(* IEC 61131-3 sources: Lasal/CPU_5344_V01/Class/Ifm2330Output, 1 file *)

(* ---- Ifm2330Output.st ---- *)
(*!
<Class
	Name               = "Ifm2330Output"
	Revision           = "0.0"
	RealtimeTask       = "false"
	CyclicTask         = "true"
	DefCyclictime      = "2 ms"
	BackgroundTask     = "false"
	Sigmatek           = "false"
	OSInterface        = "false"
	HighPriority       = "false"
	Automatic          = "false"
	UpdateMode         = "Prescan"
	SharedCommandTable = "true"
	Objectsize         = "(660,960)">
	<Channels>
		<Server Name="ActualMode" Visualized="true" Remotely="true" Initialize="false" WriteProtected="true" Retentive="false" Comment="Shows the currently active mode of the device (is only valid when the ClassState is _ClassOk and the FaultFlags are on _NoFault)"/>
		<Server Name="ClassState" Class="SDCIDevice" Visualized="true" Remotely="true" Initialize="false" WriteProtected="true" Retentive="false" Comment="Shows the current Status of the Hardware Class"/>
		<Server Name="ClassSvr" Visualized="false" Initialize="false" WriteProtected="true" Retentive="false"/>
		<Server Name="Output1" Visualized="false" Initialize="false" WriteProtected="false" Retentive="false"/>
		<Server Name="Output10" Visualized="false" Initialize="false" WriteProtected="false" Retentive="false"/>
		<Server Name="Output11" Visualized="false" Initialize="false" WriteProtected="false" Retentive="false"/>
		<Server Name="Output12" Visualized="false" Initialize="false" WriteProtected="false" Retentive="false"/>
		<Server Name="Output2" Visualized="false" Initialize="false" WriteProtected="false" Retentive="false"/>
		<Server Name="Output3" Visualized="false" Initialize="false" WriteProtected="false" Retentive="false"/>
		<Server Name="Output4" Visualized="false" Initialize="false" WriteProtected="false" Retentive="false"/>
		<Server Name="Output5" Visualized="false" Initialize="false" WriteProtected="false" Retentive="false"/>
		<Server Name="Output6" Visualized="false" Initialize="false" WriteProtected="false" Retentive="false"/>
		<Server Name="Output7" Visualized="false" Initialize="false" WriteProtected="false" Retentive="false"/>
		<Server Name="Output8" Visualized="false" Initialize="false" WriteProtected="false" Retentive="false"/>
		<Server Name="Output9" Visualized="false" Initialize="false" WriteProtected="false" Retentive="false"/>
		<Client Name="SDCIClass" Required="true" Internal="true"/>
		<Client Name="SdciIn" Required="false" Internal="false"/>
	</Channels>
	<Network Name="Ifm2330Output">
		<!-- List of Components in this network -->
		<Components>
			<Object
				Name       = "SDCIClass"
				Class      = "SDCIClassIFM2330"
				Position   = "(150,120)"
				Visualized = "true"
				Remotely   = "true">
				<Channels>
					<Server Name="ActualMode"/>
					<Server Name="ClassState"/>
					<Server Name="DeviceID"/>
					<Server Name="DirectInput"/>
					<Server Name="FaultFlags"/>
					<Server Name="Input"/>
					<Server Name="MinCycleTime"/>
					<Server Name="NbrOfEventsAvailable"/>
					<Server Name="Output"/>
					<Server Name="PortStateBits"/>
					<Server Name="VendorID"/>
					<Client Name="ReadPdoSize" Value="64"/>
					<Client Name="Required" Value="0"/>
					<Client Name="SdciIn"/>
					<Client Name="SkipEndianSwap" Value="0"/>
					<Client Name="StartUpMode" Value="_SDCI"/>
					<Client Name="WritePdoSize" Value="32"/>
				</Channels>
				<AdditionalData>
					<Entry Name="DeviceType" Value="SDCIClassIFM2330"/>
				</AdditionalData>
			</Object>
		</Components>
		<Comments>
		</Comments>
		<!-- List of Connections in this network -->
		<Connections>
			<Connection Source="SDCIClass.SdciIn" Destination="this.SdciIn" Vertices="(150,210),(38,210),"/>
			<Connection Source="this.ClassState" Destination="SDCIClass.ClassState" Vertices="(990,270),(818,210),"/>
			<Connection Source="this.SDCIClass" Destination="SDCIClass.ClassState"/>
			<Connection Source="this.ActualMode" Destination="SDCIClass.ActualMode" Vertices="(990,330),(818,450),"/>
		</Connections>
		<!-- Headerfiles -->
		<Options>
		</Options>
	</Network>
</Class>
*)
Ifm2330Output : CLASS
  //Servers:
	ClassSvr 	: SvrChCmd_DINT;
	ClassState 	: SvrChCmd_t_e_VaranErrors;
	ActualMode 	: SvrCh_t_SDCIPortMode_PTofCls_SdiasSDCIMaster;
	Output1 	: SvrCh_DINT;
	Output2 	: SvrCh_DINT;
	Output3 	: SvrCh_DINT;
	Output4 	: SvrCh_DINT;
	Output5 	: SvrCh_DINT;
	Output6 	: SvrCh_DINT;
	Output7 	: SvrCh_DINT;
	Output8 	: SvrCh_DINT;
	Output9 	: SvrCh_DINT;
	Output10 	: SvrCh_DINT;
	Output11 	: SvrCh_DINT;
	Output12 	: SvrCh_DINT;
  //Clients:
	SdciIn 	: CltChCmd_DINT;
	SDCIClass 	: CltChCmd_SDCIClassIFM2330;
  //Variables:
		bdOutputs : BDINT
		[
		];

  //Functions:

	FUNCTION VIRTUAL GLOBAL Init;

	FUNCTION VIRTUAL GLOBAL CyWork
		VAR_INPUT
			EAX 	: UDINT;
		END_VAR
		VAR_OUTPUT
			state (EAX) 	: UDINT;
		END_VAR;

	FUNCTION VIRTUAL GLOBAL ClassState::Read
		VAR_OUTPUT
			output (EAX) 	: t_e_VaranErrors;
		END_VAR;

	FUNCTION VIRTUAL GLOBAL ActualMode::Read
		VAR_OUTPUT
			output (EAX) 	: SdiasSDCIMaster::t_SDCIPortMode;
		END_VAR;
  //Tables:
	FUNCTION @STD
		VAR_OUTPUT
			ret_code	: CONFSTATES;
		END_VAR;
	FUNCTION GLOBAL TAB @CT_;
END_CLASS;

#pragma using SDCIClassIFM2330

//avdb 29092017 outputs io eiland IFM

FUNCTION VIRTUAL GLOBAL Ifm2330Output::CyWork
	VAR_INPUT
		EAX 	: UDINT;
	END_VAR
	VAR_OUTPUT
		state (EAX) 	: UDINT;
	END_VAR

  // get outputs from servers
  bdOutputs.25 := Output1=1;
  bdOutputs.9 := Output2=1;
  bdOutputs.17 := Output3=1;
  bdOutputs.1 := Output4=1;
  bdOutputs.26 := Output5=1;
  bdOutputs.10 := Output6=1;
  bdOutputs.18 := Output7=1;
  bdOutputs.2 := Output8=1;
  bdOutputs.27 := Output9=1;
  bdOutputs.11 := Output10=1;
  bdOutputs.19 := Output11=1;
  bdOutputs.3 := Output12=1;

  // and write outputs to ifm splitterbox
  SDCIClass.SetWritePdoDWord(WriteValue:=bdOutputs, WriteOffset:=0);

	state := READY;

END_FUNCTION

FUNCTION VIRTUAL GLOBAL Ifm2330Output::Init

END_FUNCTION

FUNCTION VIRTUAL GLOBAL Ifm2330Output::ClassState::Read
	VAR_OUTPUT
		output (EAX) 	: t_e_VaranErrors;
	END_VAR

	ClassState := SDCIClass.ClassState.Read();
	output := ClassState;

END_FUNCTION

FUNCTION VIRTUAL GLOBAL Ifm2330Output::ActualMode::Read
	VAR_OUTPUT
		output (EAX) 	: SdiasSDCIMaster::t_SDCIPortMode;
	END_VAR

	ActualMode := SDCIClass.ActualMode.Read();
	output := ActualMode;

END_FUNCTION
